# B&R Automation Studio project DuctLines (part 12)

#### Cyclic.ld
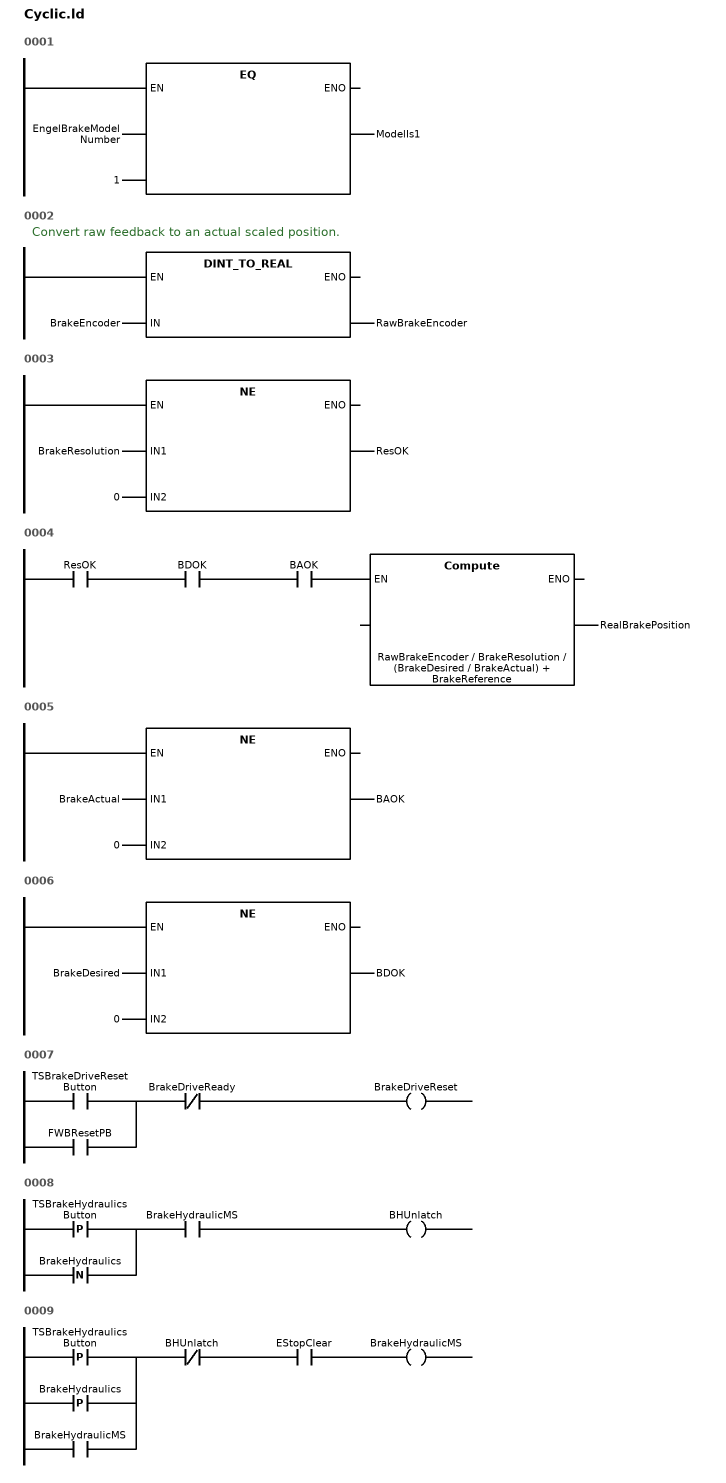
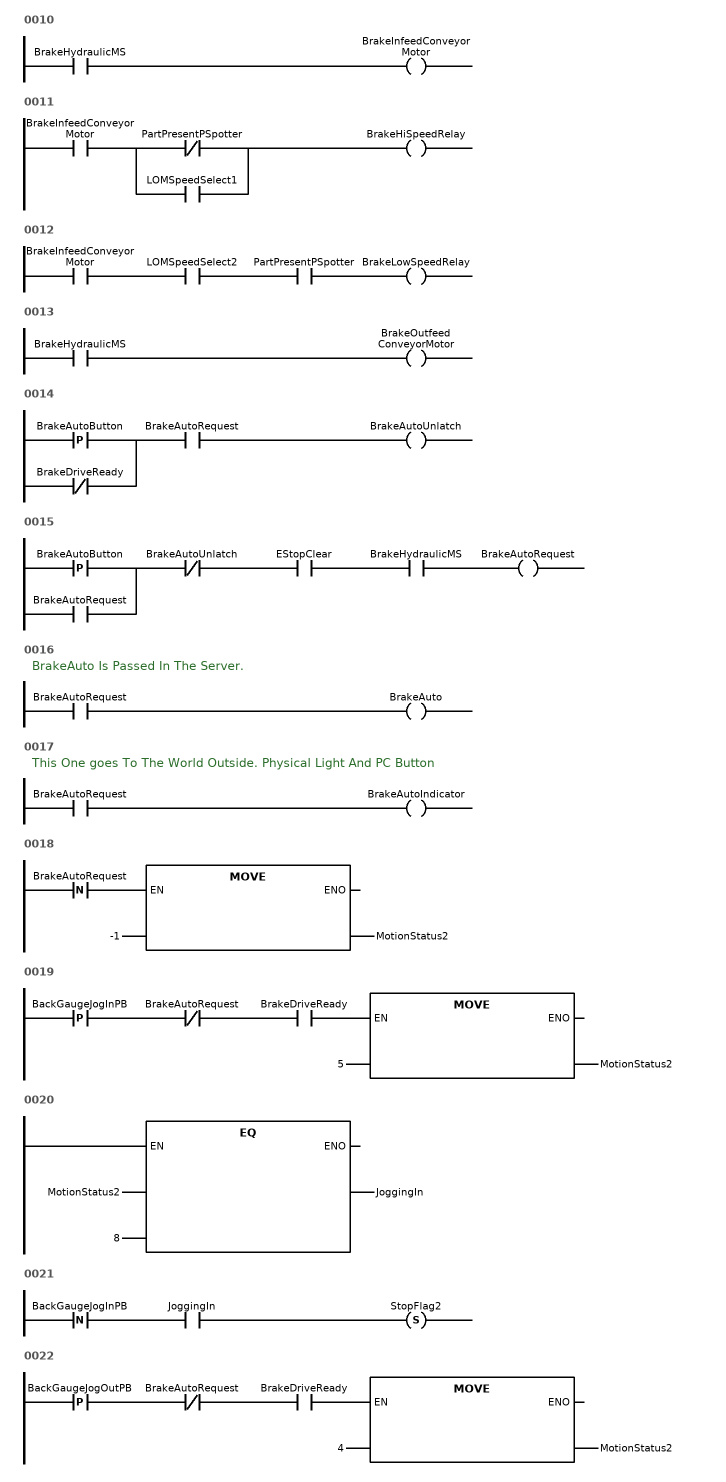
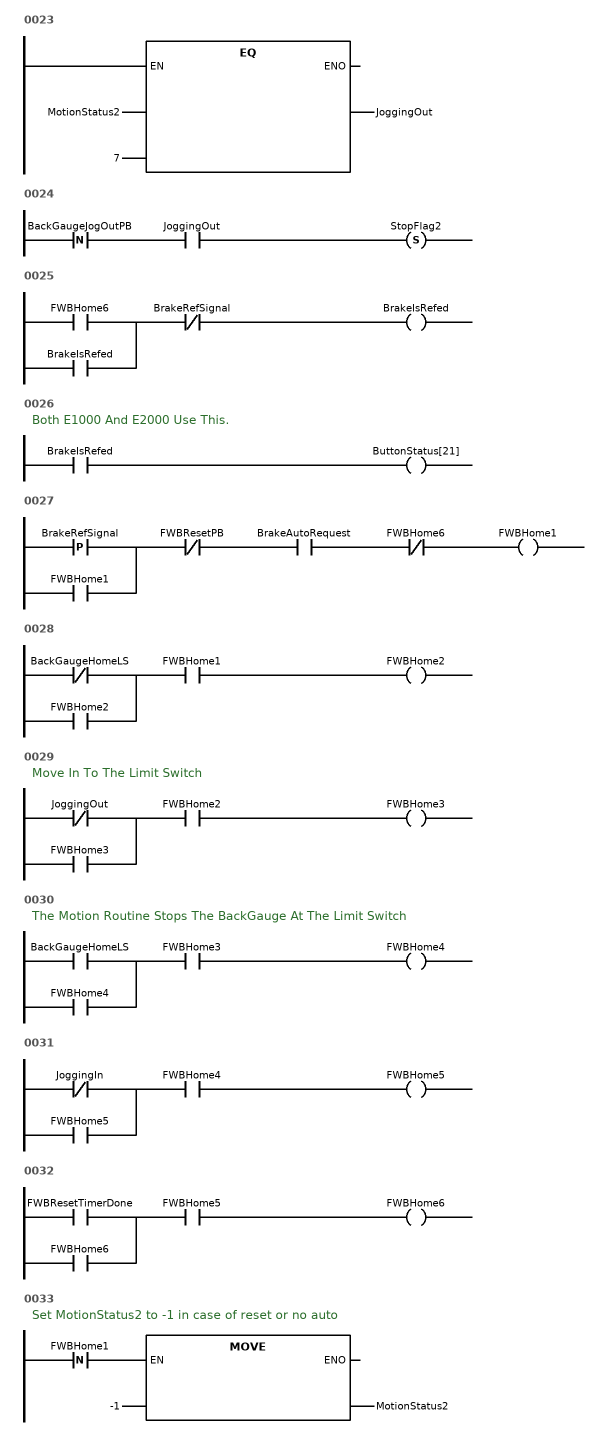
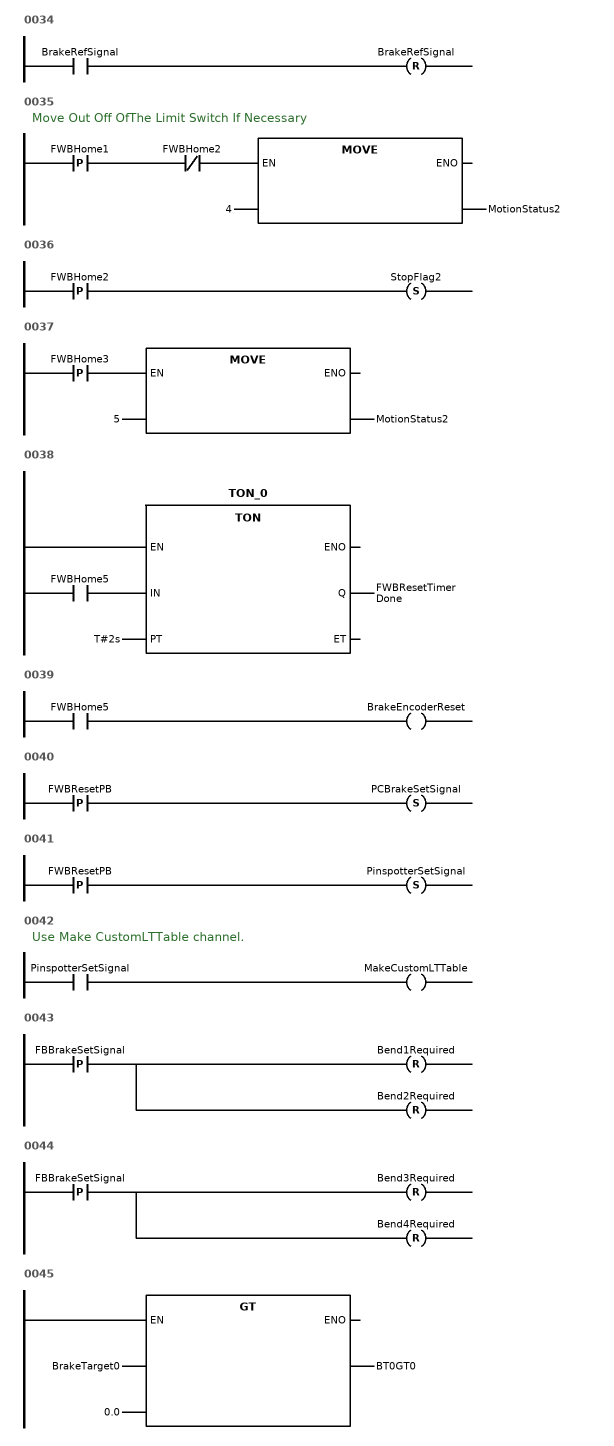
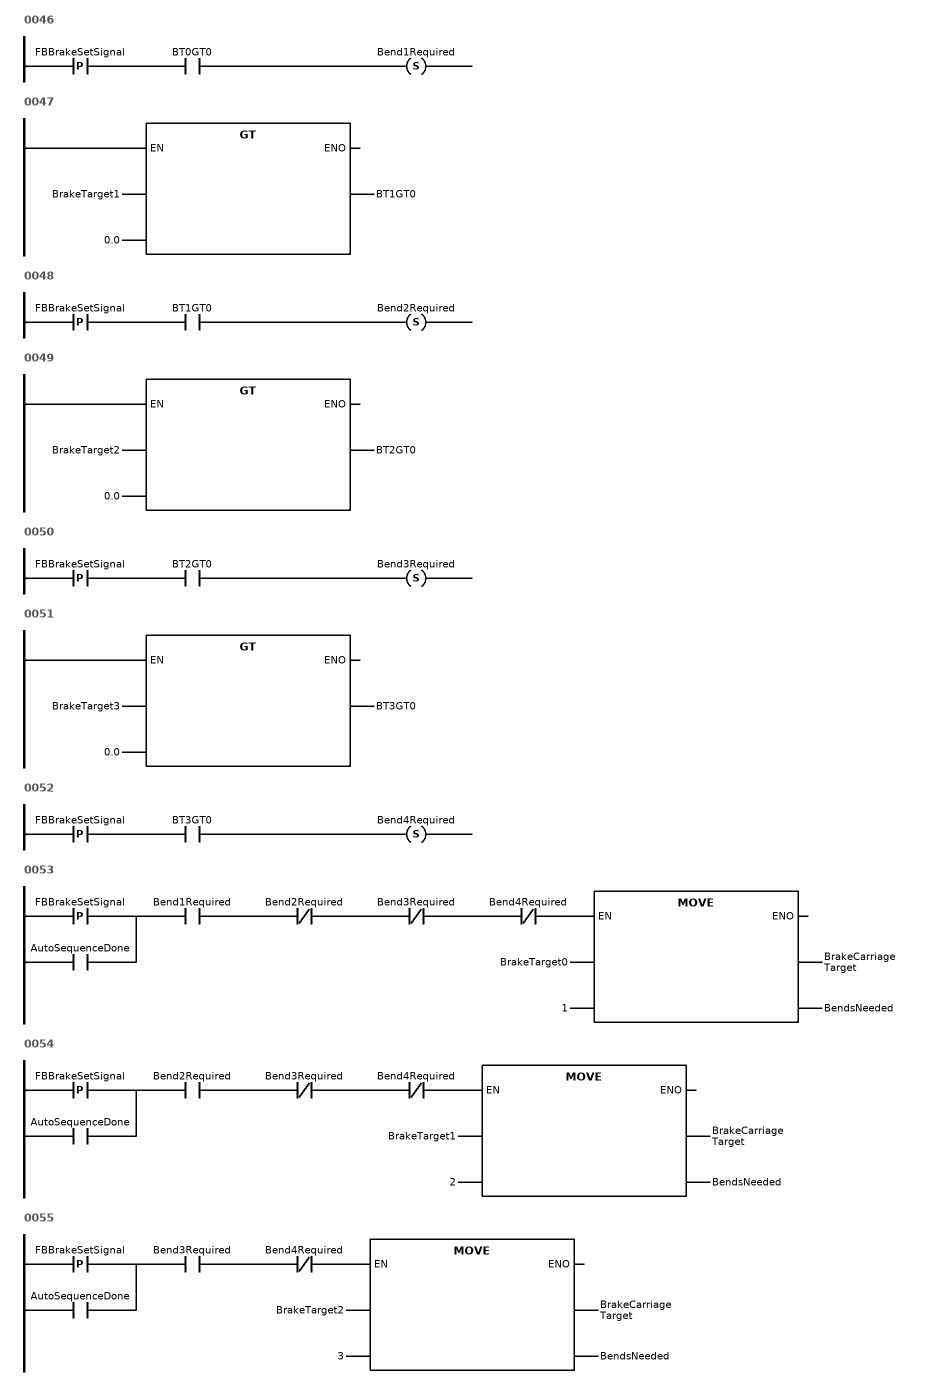
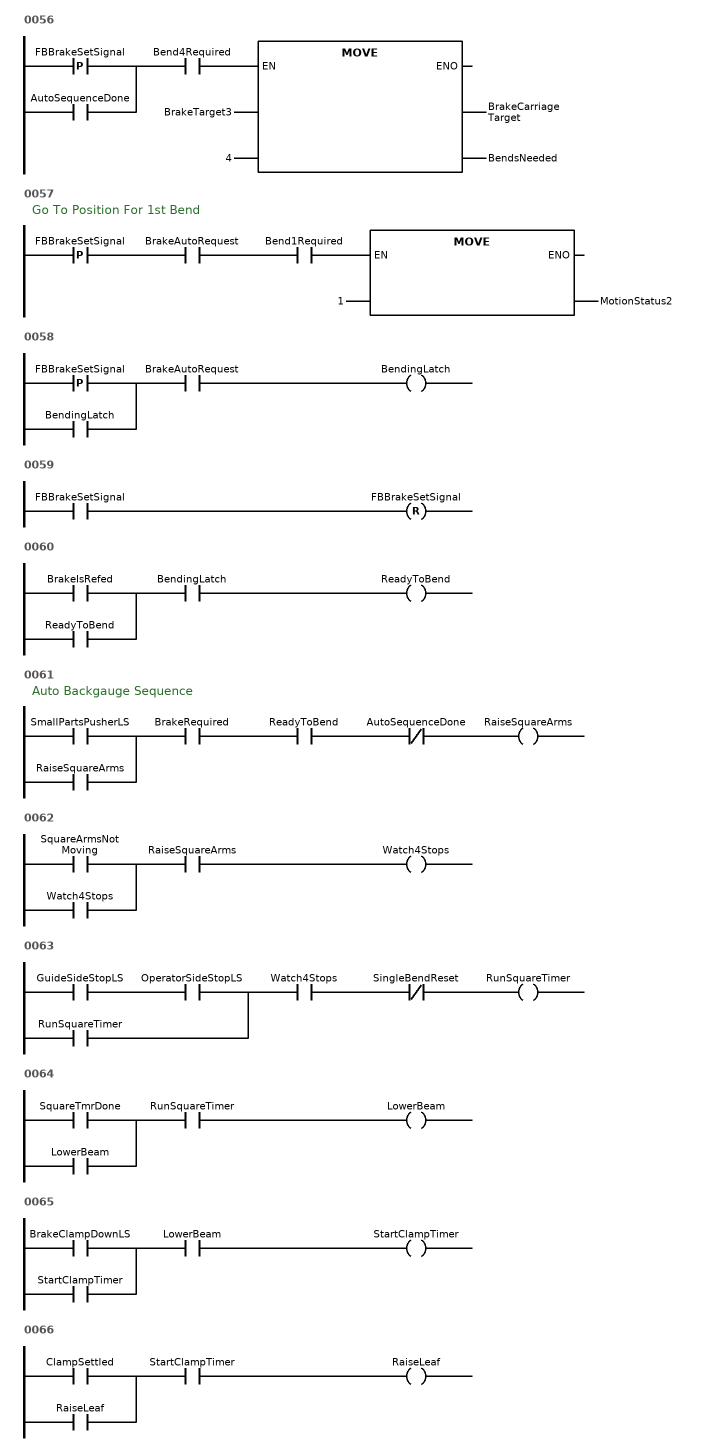
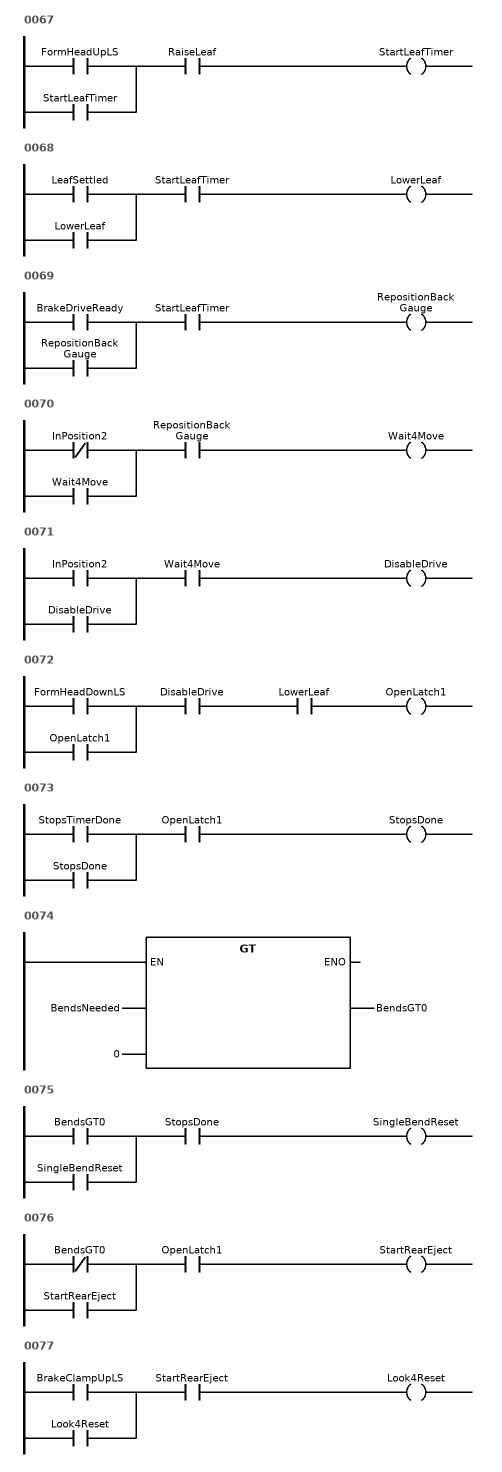
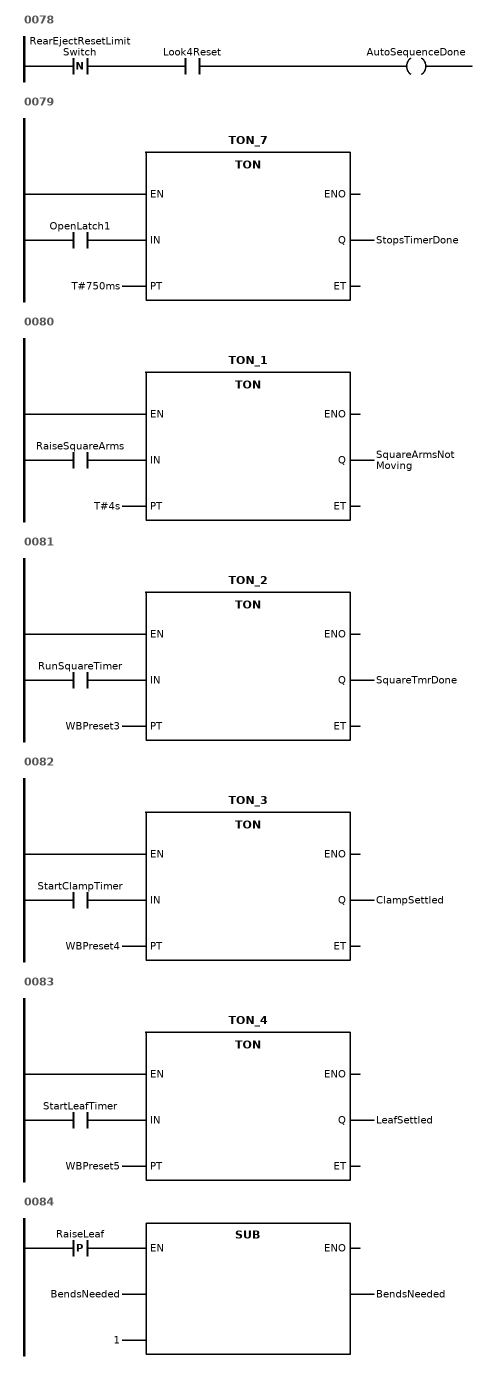
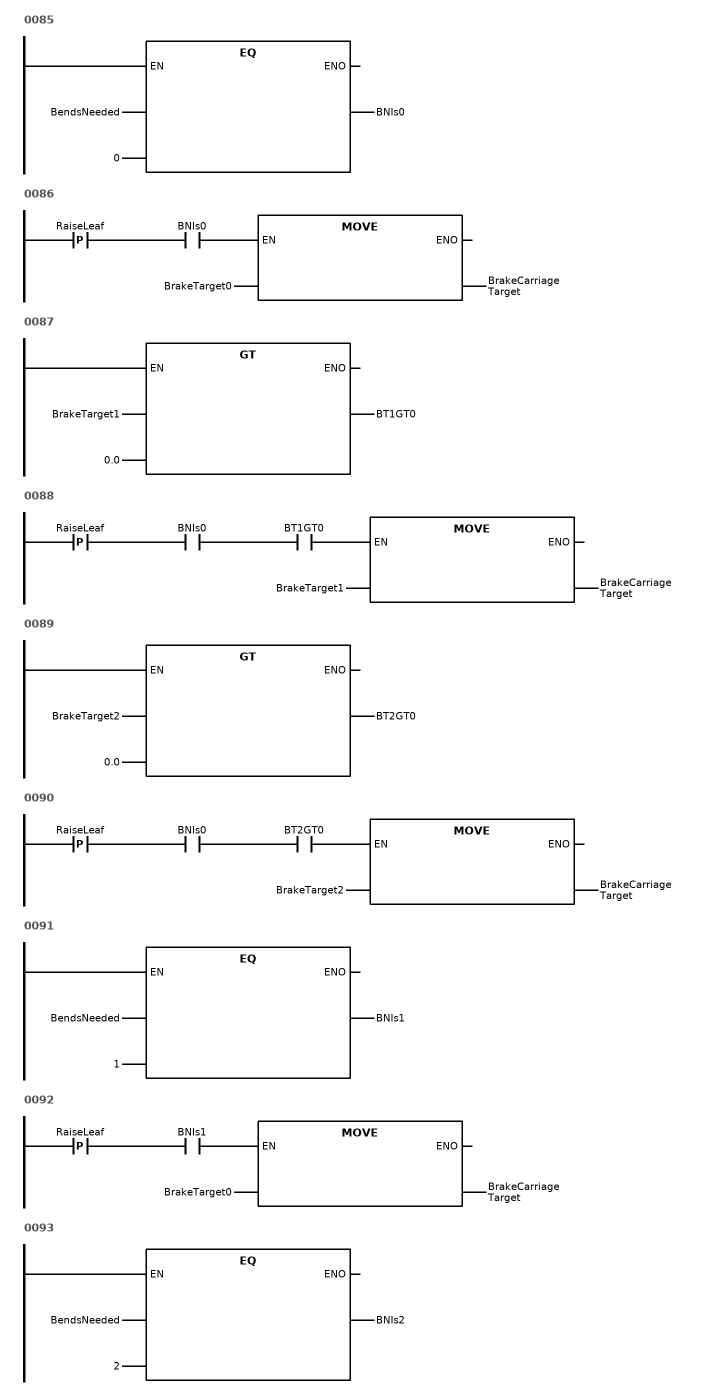
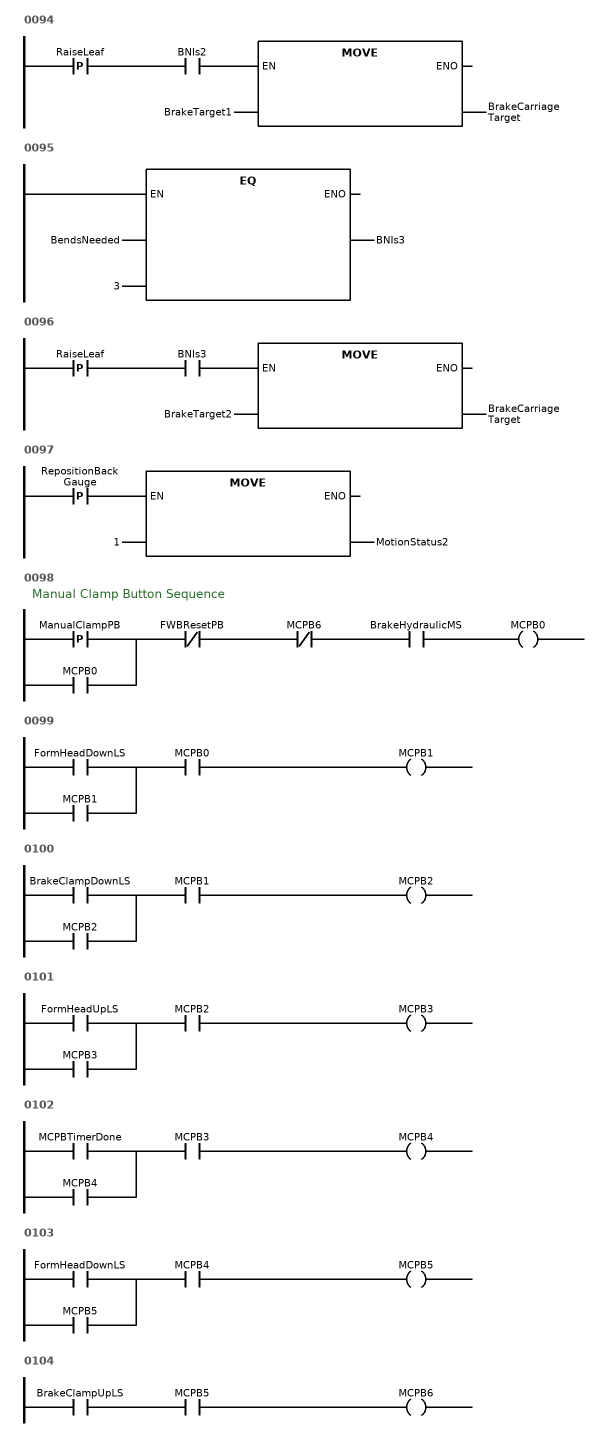
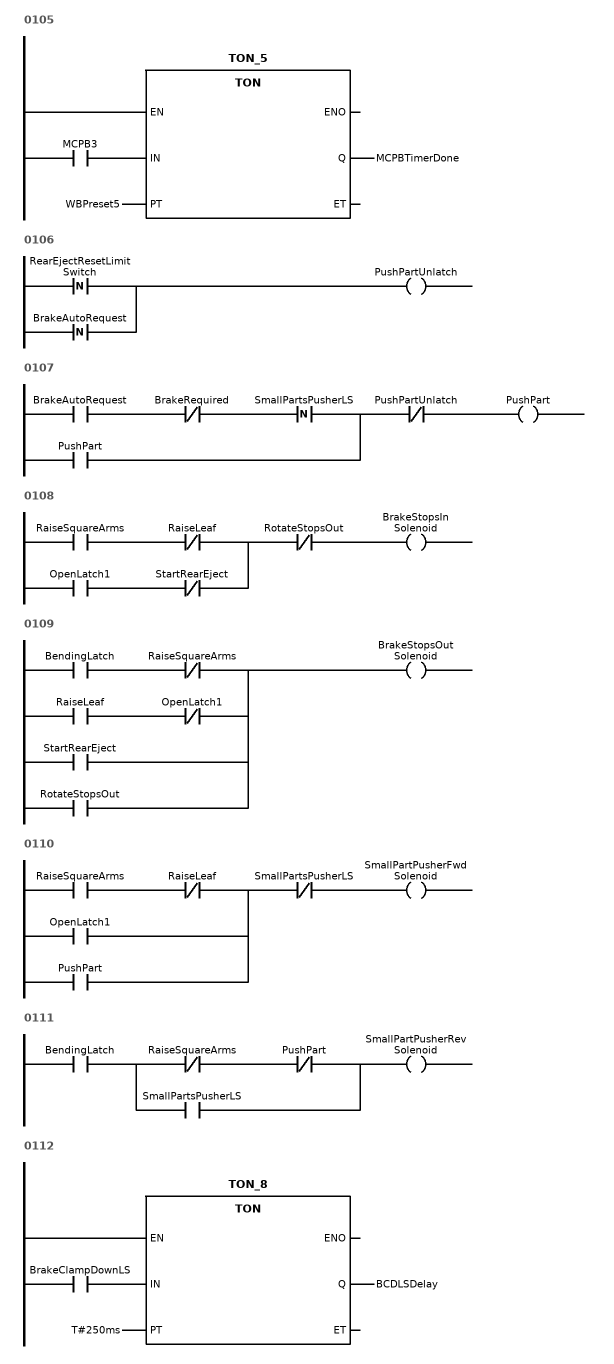
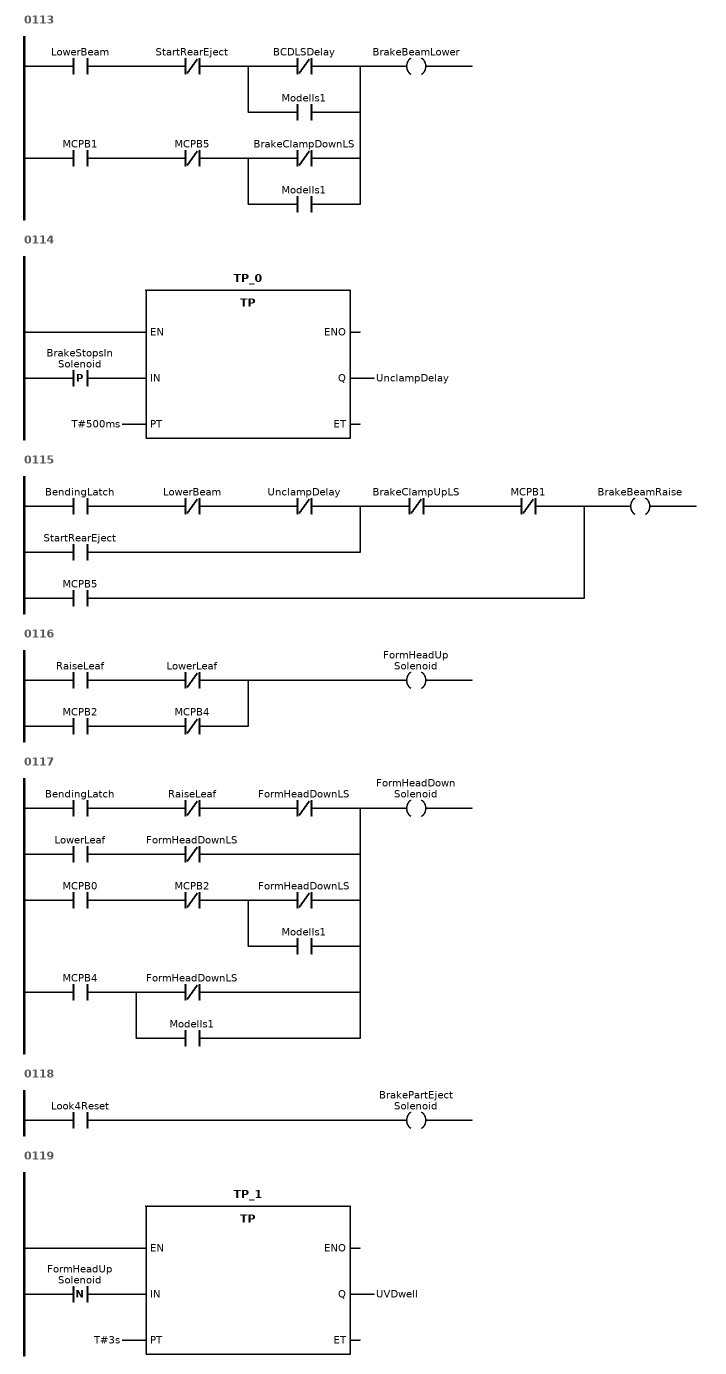
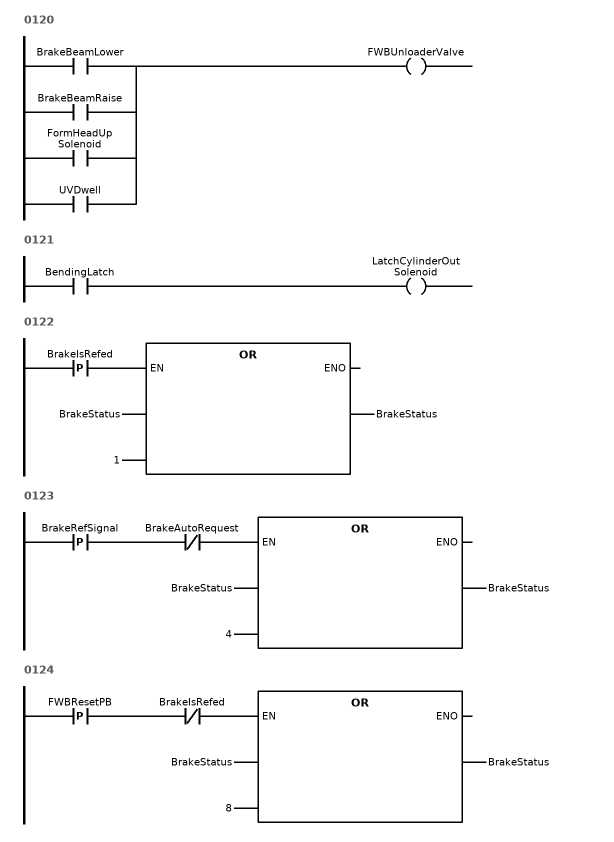
Ladder, written as Structured Text:
```iecst
PROGRAM _CYCLIC
VAR
    _e1 : R_TRIG;
    _e2 : F_TRIG;
    _e3 : R_TRIG;
    _e4 : R_TRIG;
    _e5 : R_TRIG;
    _e6 : R_TRIG;
    _e7 : F_TRIG;
    _e8 : R_TRIG;
    _e9 : F_TRIG;
    _e10 : R_TRIG;
    _e11 : F_TRIG;
    _e12 : R_TRIG;
    _e13 : F_TRIG;
    _e14 : R_TRIG;
    _e15 : R_TRIG;
    _e16 : R_TRIG;
    _e17 : R_TRIG;
    _e18 : R_TRIG;
    _e19 : R_TRIG;
    _e20 : R_TRIG;
    _e21 : R_TRIG;
    _e22 : R_TRIG;
    _e23 : R_TRIG;
    _e24 : R_TRIG;
    _e25 : R_TRIG;
    _p26 : BOOL;
    _e27 : R_TRIG;
    _p28 : BOOL;
    _e29 : R_TRIG;
    _p30 : BOOL;
    _e31 : R_TRIG;
    _e32 : R_TRIG;
    _e33 : R_TRIG;
    _e34 : F_TRIG;
    _e35 : R_TRIG;
    _e36 : R_TRIG;
    _e37 : R_TRIG;
    _e38 : R_TRIG;
    _e39 : R_TRIG;
    _e40 : R_TRIG;
    _e41 : R_TRIG;
    _e42 : R_TRIG;
    _e43 : R_TRIG;
    _e44 : F_TRIG;
    _e45 : F_TRIG;
    _e46 : F_TRIG;
    _e47 : R_TRIG;
    _e48 : F_TRIG;
    _e49 : R_TRIG;
    _e50 : R_TRIG;
    _e51 : R_TRIG;
END_VAR
(* Network 1 *)
ModelIs1 := EngelBrakeModelNumber = 1;

(* Network 2: Convert raw feedback to an actual scaled position. *)
RawBrakeEncoder := DINT_TO_REAL(BrakeEncoder);

(* Network 3 *)
ResOK := BrakeResolution <> 0;

(* Network 4 *)
IF ResOK AND BDOK AND BAOK THEN
    RealBrakePosition := RawBrakeEncoder / BrakeResolution / (BrakeDesired / BrakeActual) + BrakeReference;
END_IF;

(* Network 5 *)
BAOK := BrakeActual <> 0;

(* Network 6 *)
BDOK := BrakeDesired <> 0;

(* Network 7 *)
BrakeDriveReset := (TSBrakeDriveResetButton OR FWBResetPB) AND NOT BrakeDriveReady;

(* Network 8 *)
_e1(CLK := TSBrakeHydraulicsButton);
_e2(CLK := BrakeHydraulics);
BHUnlatch := (_e1.Q OR _e2.Q) AND BrakeHydraulicMS;

(* Network 9 *)
_e3(CLK := TSBrakeHydraulicsButton);
_e4(CLK := BrakeHydraulics);
BrakeHydraulicMS := (_e3.Q OR _e4.Q OR BrakeHydraulicMS) AND NOT BHUnlatch AND EStopClear;

(* Network 10 *)
BrakeInfeedConveyorMotor := BrakeHydraulicMS;

(* Network 11 *)
BrakeHiSpeedRelay := BrakeInfeedConveyorMotor AND (NOT PartPresentPSpotter OR LOMSpeedSelect1);

(* Network 12 *)
BrakeLowSpeedRelay := BrakeInfeedConveyorMotor AND LOMSpeedSelect2 AND PartPresentPSpotter;

(* Network 13 *)
BrakeOutfeedConveyorMotor := BrakeHydraulicMS;

(* Network 14 *)
_e5(CLK := BrakeAutoButton);
BrakeAutoUnlatch := (_e5.Q OR NOT BrakeDriveReady) AND BrakeAutoRequest;

(* Network 15 *)
_e6(CLK := BrakeAutoButton);
BrakeAutoRequest := (_e6.Q OR BrakeAutoRequest) AND NOT BrakeAutoUnlatch AND EStopClear AND BrakeHydraulicMS;

(* Network 16: BrakeAuto Is Passed In The Server. *)
BrakeAuto := BrakeAutoRequest;

(* Network 17: This One goes To The World Outside. Physical Light And PC Button *)
BrakeAutoIndicator := BrakeAutoRequest;

(* Network 18 *)
_e7(CLK := BrakeAutoRequest);
IF _e7.Q THEN MotionStatus2 := -1; END_IF;

(* Network 19 *)
_e8(CLK := BackGaugeJogInPB);
IF _e8.Q AND NOT BrakeAutoRequest AND BrakeDriveReady THEN MotionStatus2 := 5; END_IF;

(* Network 20 *)
JoggingIn := MotionStatus2 = 8;

(* Network 21 *)
_e9(CLK := BackGaugeJogInPB);
IF _e9.Q AND JoggingIn THEN StopFlag2 := TRUE; END_IF;

(* Network 22 *)
_e10(CLK := BackGaugeJogOutPB);
IF _e10.Q AND NOT BrakeAutoRequest AND BrakeDriveReady THEN MotionStatus2 := 4; END_IF;

(* Network 23 *)
JoggingOut := MotionStatus2 = 7;

(* Network 24 *)
_e11(CLK := BackGaugeJogOutPB);
IF _e11.Q AND JoggingOut THEN StopFlag2 := TRUE; END_IF;

(* Network 25 *)
BrakeIsRefed := (FWBHome6 OR BrakeIsRefed) AND NOT BrakeRefSignal;

(* Network 26: Both E1000 And E2000 Use This. *)
ButtonStatus[21] := BrakeIsRefed;

(* Network 27 *)
_e12(CLK := BrakeRefSignal);
FWBHome1 := (_e12.Q OR FWBHome1) AND NOT FWBResetPB AND BrakeAutoRequest AND NOT FWBHome6;

(* Network 28 *)
FWBHome2 := (NOT BackGaugeHomeLS OR FWBHome2) AND FWBHome1;

(* Network 29: Move In To The Limit Switch *)
FWBHome3 := (NOT JoggingOut OR FWBHome3) AND FWBHome2;

(* Network 30: The Motion Routine Stops The BackGauge At The Limit Switch *)
FWBHome4 := (BackGaugeHomeLS OR FWBHome4) AND FWBHome3;

(* Network 31 *)
FWBHome5 := (NOT JoggingIn OR FWBHome5) AND FWBHome4;

(* Network 32 *)
FWBHome6 := (FWBResetTimerDone OR FWBHome6) AND FWBHome5;

(* Network 33: Set MotionStatus2 to -1 in case of reset or no auto *)
_e13(CLK := FWBHome1);
IF _e13.Q THEN MotionStatus2 := -1; END_IF;

(* Network 34 *)
IF BrakeRefSignal THEN BrakeRefSignal := FALSE; END_IF;

(* Network 35: Move Out Off OfThe Limit Switch If Necessary *)
_e14(CLK := FWBHome1);
IF _e14.Q AND NOT FWBHome2 THEN MotionStatus2 := 4; END_IF;

(* Network 36 *)
_e15(CLK := FWBHome2);
IF _e15.Q THEN StopFlag2 := TRUE; END_IF;

(* Network 37 *)
_e16(CLK := FWBHome3);
IF _e16.Q THEN MotionStatus2 := 5; END_IF;

(* Network 38 *)
TON_0(IN := FWBHome5, PT := T#2s);
FWBResetTimerDone := TON_0.Q;

(* Network 39 *)
BrakeEncoderReset := FWBHome5;

(* Network 40 *)
_e17(CLK := FWBResetPB);
IF _e17.Q THEN PCBrakeSetSignal := TRUE; END_IF;

(* Network 41 *)
_e18(CLK := FWBResetPB);
IF _e18.Q THEN PinspotterSetSignal := TRUE; END_IF;

(* Network 42: Use Make CustomLTTable channel. *)
MakeCustomLTTable := PinspotterSetSignal;

(* Network 43 *)
_e19(CLK := FBBrakeSetSignal);
IF _e19.Q THEN
    Bend1Required := FALSE;
    Bend2Required := FALSE;
END_IF;

(* Network 44 *)
_e20(CLK := FBBrakeSetSignal);
IF _e20.Q THEN
    Bend3Required := FALSE;
    Bend4Required := FALSE;
END_IF;

(* Network 45 *)
BT0GT0 := BrakeTarget0 > 0.0;

(* Network 46 *)
_e21(CLK := FBBrakeSetSignal);
IF _e21.Q AND BT0GT0 THEN Bend1Required := TRUE; END_IF;

(* Network 47 *)
BT1GT0 := BrakeTarget1 > 0.0;

(* Network 48 *)
_e22(CLK := FBBrakeSetSignal);
IF _e22.Q AND BT1GT0 THEN Bend2Required := TRUE; END_IF;

(* Network 49 *)
BT2GT0 := BrakeTarget2 > 0.0;

(* Network 50 *)
_e23(CLK := FBBrakeSetSignal);
IF _e23.Q AND BT2GT0 THEN Bend3Required := TRUE; END_IF;

(* Network 51 *)
BT3GT0 := BrakeTarget3 > 0.0;

(* Network 52 *)
_e24(CLK := FBBrakeSetSignal);
IF _e24.Q AND BT3GT0 THEN Bend4Required := TRUE; END_IF;

(* Network 53 *)
_e25(CLK := FBBrakeSetSignal);
_p26 := (_e25.Q OR AutoSequenceDone) AND Bend1Required AND NOT Bend2Required AND NOT Bend3Required AND NOT Bend4Required;
IF _p26 THEN
    BrakeCarriageTarget := BrakeTarget0;
    BendsNeeded := 1;
END_IF;

(* Network 54 *)
_e27(CLK := FBBrakeSetSignal);
_p28 := (_e27.Q OR AutoSequenceDone) AND Bend2Required AND NOT Bend3Required AND NOT Bend4Required;
IF _p28 THEN
    BrakeCarriageTarget := BrakeTarget1;
    BendsNeeded := 2;
END_IF;

(* Network 55 *)
_e29(CLK := FBBrakeSetSignal);
_p30 := (_e29.Q OR AutoSequenceDone) AND Bend3Required AND NOT Bend4Required;
IF _p30 THEN
    BrakeCarriageTarget := BrakeTarget2;
    BendsNeeded := 3;
END_IF;

(* Network 56 *)
_e31(CLK := FBBrakeSetSignal);
IF (_e31.Q OR AutoSequenceDone) AND Bend4Required THEN
    BrakeCarriageTarget := BrakeTarget3;
    BendsNeeded := 4;
END_IF;

(* Network 57: Go To Position For 1st Bend *)
_e32(CLK := FBBrakeSetSignal);
IF _e32.Q AND BrakeAutoRequest AND Bend1Required THEN MotionStatus2 := 1; END_IF;

(* Network 58 *)
_e33(CLK := FBBrakeSetSignal);
BendingLatch := (_e33.Q OR BendingLatch) AND BrakeAutoRequest;

(* Network 59 *)
IF FBBrakeSetSignal THEN FBBrakeSetSignal := FALSE; END_IF;

(* Network 60 *)
ReadyToBend := (BrakeIsRefed OR ReadyToBend) AND BendingLatch;

(* Network 61: Auto Backgauge Sequence *)
RaiseSquareArms := (SmallPartsPusherLS OR RaiseSquareArms) AND BrakeRequired AND ReadyToBend AND NOT AutoSequenceDone;

(* Network 62 *)
Watch4Stops := (SquareArmsNotMoving OR Watch4Stops) AND RaiseSquareArms;

(* Network 63 *)
RunSquareTimer := ((GuideSideStopLS AND OperatorSideStopLS) OR RunSquareTimer) AND Watch4Stops AND NOT SingleBendReset;

(* Network 64 *)
LowerBeam := (SquareTmrDone OR LowerBeam) AND RunSquareTimer;

(* Network 65 *)
StartClampTimer := (BrakeClampDownLS OR StartClampTimer) AND LowerBeam;

(* Network 66 *)
RaiseLeaf := (ClampSettled OR RaiseLeaf) AND StartClampTimer;

(* Network 67 *)
StartLeafTimer := (FormHeadUpLS OR StartLeafTimer) AND RaiseLeaf;

(* Network 68 *)
LowerLeaf := (LeafSettled OR LowerLeaf) AND StartLeafTimer;

(* Network 69 *)
RepositionBackGauge := (BrakeDriveReady OR RepositionBackGauge) AND StartLeafTimer;

(* Network 70 *)
Wait4Move := (NOT InPosition2 OR Wait4Move) AND RepositionBackGauge;

(* Network 71 *)
DisableDrive := (InPosition2 OR DisableDrive) AND Wait4Move;

(* Network 72 *)
OpenLatch1 := (FormHeadDownLS OR OpenLatch1) AND DisableDrive AND LowerLeaf;

(* Network 73 *)
StopsDone := (StopsTimerDone OR StopsDone) AND OpenLatch1;

(* Network 74 *)
BendsGT0 := BendsNeeded > 0;

(* Network 75 *)
SingleBendReset := (BendsGT0 OR SingleBendReset) AND StopsDone;

(* Network 76 *)
StartRearEject := (NOT BendsGT0 OR StartRearEject) AND OpenLatch1;

(* Network 77 *)
Look4Reset := (BrakeClampUpLS OR Look4Reset) AND StartRearEject;

(* Network 78 *)
_e34(CLK := RearEjectResetLimitSwitch);
AutoSequenceDone := _e34.Q AND Look4Reset;

(* Network 79 *)
TON_7(IN := OpenLatch1, PT := T#750ms);
StopsTimerDone := TON_7.Q;

(* Network 80 *)
TON_1(IN := RaiseSquareArms, PT := T#4s);
SquareArmsNotMoving := TON_1.Q;

(* Network 81 *)
TON_2(IN := RunSquareTimer, PT := WBPreset3);
SquareTmrDone := TON_2.Q;

(* Network 82 *)
TON_3(IN := StartClampTimer, PT := WBPreset4);
ClampSettled := TON_3.Q;

(* Network 83 *)
TON_4(IN := StartLeafTimer, PT := WBPreset5);
LeafSettled := TON_4.Q;

(* Network 84 *)
_e35(CLK := RaiseLeaf);
IF _e35.Q THEN BendsNeeded := BendsNeeded - 1; END_IF;

(* Network 85 *)
BNIs0 := BendsNeeded = 0;

(* Network 86 *)
_e36(CLK := RaiseLeaf);
IF _e36.Q AND BNIs0 THEN BrakeCarriageTarget := BrakeTarget0; END_IF;

(* Network 87 *)
BT1GT0 := BrakeTarget1 > 0.0;

(* Network 88 *)
_e37(CLK := RaiseLeaf);
IF _e37.Q AND BNIs0 AND BT1GT0 THEN BrakeCarriageTarget := BrakeTarget1; END_IF;

(* Network 89 *)
BT2GT0 := BrakeTarget2 > 0.0;

(* Network 90 *)
_e38(CLK := RaiseLeaf);
IF _e38.Q AND BNIs0 AND BT2GT0 THEN BrakeCarriageTarget := BrakeTarget2; END_IF;

(* Network 91 *)
BNIs1 := BendsNeeded = 1;

(* Network 92 *)
_e39(CLK := RaiseLeaf);
IF _e39.Q AND BNIs1 THEN BrakeCarriageTarget := BrakeTarget0; END_IF;

(* Network 93 *)
BNIs2 := BendsNeeded = 2;

(* Network 94 *)
_e40(CLK := RaiseLeaf);
IF _e40.Q AND BNIs2 THEN BrakeCarriageTarget := BrakeTarget1; END_IF;

(* Network 95 *)
BNIs3 := BendsNeeded = 3;

(* Network 96 *)
_e41(CLK := RaiseLeaf);
IF _e41.Q AND BNIs3 THEN BrakeCarriageTarget := BrakeTarget2; END_IF;

(* Network 97 *)
_e42(CLK := RepositionBackGauge);
IF _e42.Q THEN MotionStatus2 := 1; END_IF;

(* Network 98: Manual Clamp Button Sequence *)
_e43(CLK := ManualClampPB);
MCPB0 := (_e43.Q OR MCPB0) AND NOT FWBResetPB AND NOT MCPB6 AND BrakeHydraulicMS;

(* Network 99 *)
MCPB1 := (FormHeadDownLS OR MCPB1) AND MCPB0;

(* Network 100 *)
MCPB2 := (BrakeClampDownLS OR MCPB2) AND MCPB1;

(* Network 101 *)
MCPB3 := (FormHeadUpLS OR MCPB3) AND MCPB2;

(* Network 102 *)
MCPB4 := (MCPBTimerDone OR MCPB4) AND MCPB3;

(* Network 103 *)
MCPB5 := (FormHeadDownLS OR MCPB5) AND MCPB4;

(* Network 104 *)
MCPB6 := BrakeClampUpLS AND MCPB5;

(* Network 105 *)
TON_5(IN := MCPB3, PT := WBPreset5);
MCPBTimerDone := TON_5.Q;

(* Network 106 *)
_e44(CLK := RearEjectResetLimitSwitch);
_e45(CLK := BrakeAutoRequest);
PushPartUnlatch := _e44.Q OR _e45.Q;

(* Network 107 *)
_e46(CLK := SmallPartsPusherLS);
PushPart := ((BrakeAutoRequest AND NOT BrakeRequired AND _e46.Q) OR PushPart) AND NOT PushPartUnlatch;

(* Network 108 *)
BrakeStopsInSolenoid := ((RaiseSquareArms AND NOT RaiseLeaf) OR (OpenLatch1 AND NOT StartRearEject)) AND NOT RotateStopsOut;

(* Network 109 *)
BrakeStopsOutSolenoid := (BendingLatch AND NOT RaiseSquareArms) OR (RaiseLeaf AND NOT OpenLatch1) OR StartRearEject OR RotateStopsOut;

(* Network 110 *)
SmallPartPusherFwdSolenoid := ((RaiseSquareArms AND NOT RaiseLeaf) OR OpenLatch1 OR PushPart) AND NOT SmallPartsPusherLS;

(* Network 111 *)
SmallPartPusherRevSolenoid := BendingLatch AND ((NOT RaiseSquareArms AND NOT PushPart) OR SmallPartsPusherLS);

(* Network 112 *)
TON_8(IN := BrakeClampDownLS, PT := T#250ms);
BCDLSDelay := TON_8.Q;

(* Network 113 *)
BrakeBeamLower := (LowerBeam AND NOT StartRearEject AND (NOT BCDLSDelay OR ModelIs1)) OR (MCPB1 AND NOT MCPB5 AND (NOT BrakeClampDownLS OR ModelIs1));

(* Network 114 *)
_e47(CLK := BrakeStopsInSolenoid);
TP_0(IN := _e47.Q, PT := T#500ms);
UnclampDelay := TP_0.Q;

(* Network 115 *)
BrakeBeamRaise := (((BendingLatch AND NOT LowerBeam AND NOT UnclampDelay) OR StartRearEject) AND NOT BrakeClampUpLS AND NOT MCPB1) OR MCPB5;

(* Network 116 *)
FormHeadUpSolenoid := (RaiseLeaf AND NOT LowerLeaf) OR (MCPB2 AND NOT MCPB4);

(* Network 117 *)
FormHeadDownSolenoid := (BendingLatch AND NOT RaiseLeaf AND NOT FormHeadDownLS) OR (LowerLeaf AND NOT FormHeadDownLS) OR (MCPB0 AND NOT MCPB2 AND (NOT FormHeadDownLS OR ModelIs1)) OR (MCPB4 AND (NOT FormHeadDownLS OR ModelIs1));

(* Network 118 *)
BrakePartEjectSolenoid := Look4Reset;

(* Network 119 *)
_e48(CLK := FormHeadUpSolenoid);
TP_1(IN := _e48.Q, PT := T#3s);
UVDwell := TP_1.Q;

(* Network 120 *)
FWBUnloaderValve := BrakeBeamLower OR BrakeBeamRaise OR FormHeadUpSolenoid OR UVDwell;

(* Network 121 *)
LatchCylinderOutSolenoid := BendingLatch;

(* Network 122 *)
_e49(CLK := BrakeIsRefed);
IF _e49.Q THEN BrakeStatus := BrakeStatus OR 1; END_IF;

(* Network 123 *)
_e50(CLK := BrakeRefSignal);
IF _e50.Q AND NOT BrakeAutoRequest THEN BrakeStatus := BrakeStatus OR 4; END_IF;

(* Network 124 *)
_e51(CLK := FWBResetPB);
IF _e51.Q AND NOT BrakeIsRefed THEN BrakeStatus := BrakeStatus OR 8; END_IF;
END_PROGRAM
```

#### Init.ld
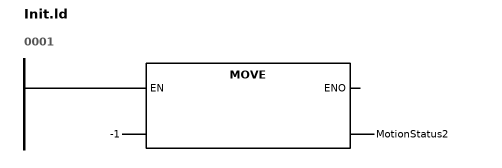
Ladder, written as Structured Text:
```iecst
PROGRAM _INIT
(* Network 1 *)
MotionStatus2 := -1;
END_PROGRAM
```

### Program Logical/PMaster (IEC)

#### Variables.var
```iecst
VAR
	PunchCurrentSelect : DINT;
	OGResult : DINT;
	OGLatch : BOOL;
	FourFootCoil : BOOL;
	FiveFootCoil : BOOL;
	SixFootCoil : BOOL;
	FourResult : DINT;
	FFCLatch : BOOL;
	OneResult : DINT;
	OutsideLatch : BOOL;
	DamperResult : DINT;
	DamperLatch : BOOL;
END_VAR
```

#### Cyclic.ld
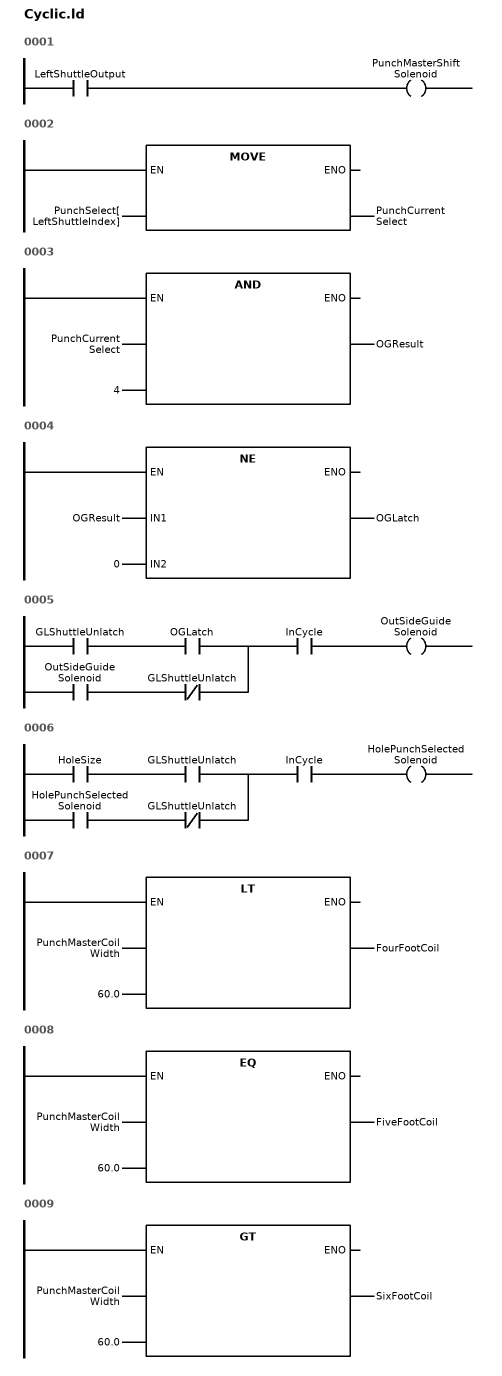
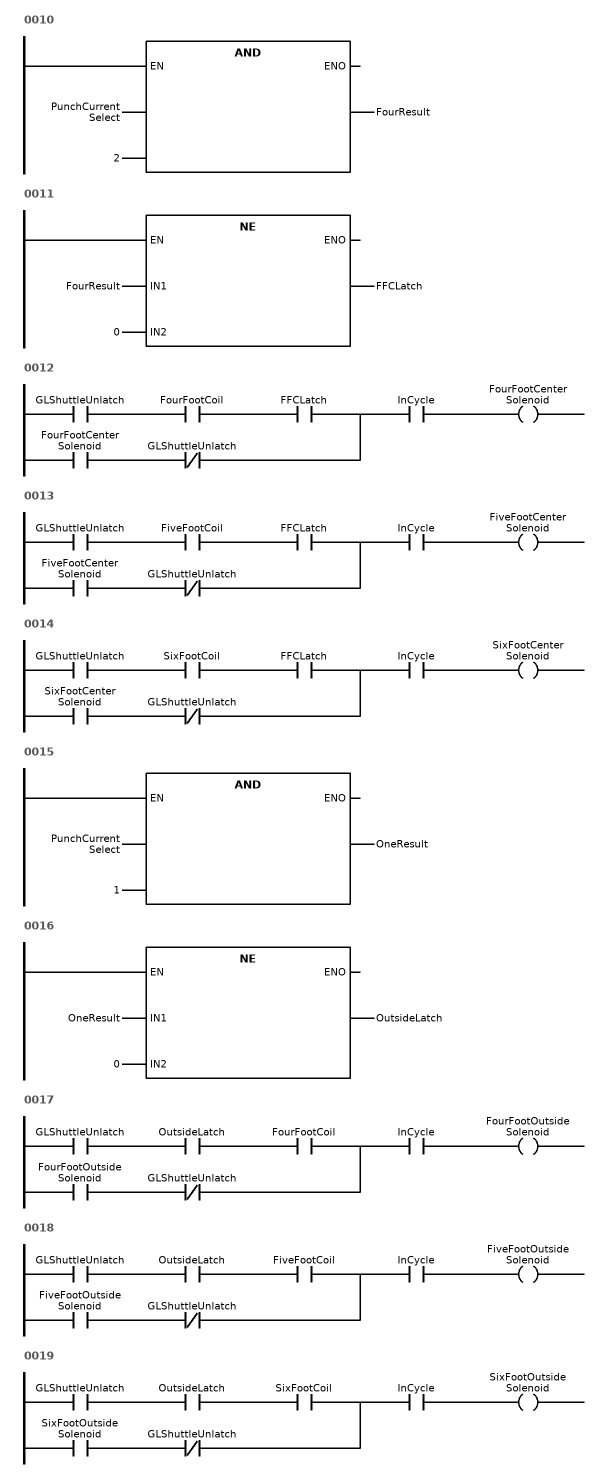
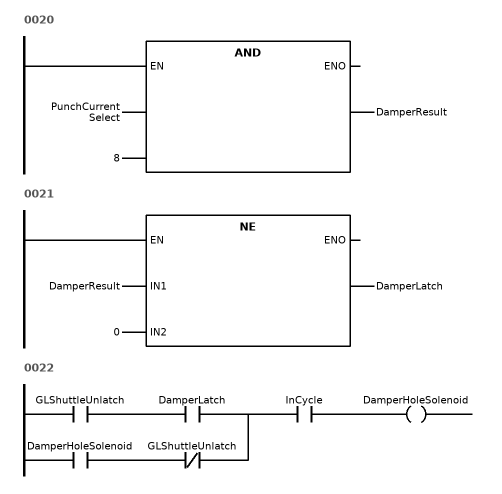
Ladder, written as Structured Text:
```iecst
PROGRAM _CYCLIC
(* Network 1 *)
PunchMasterShiftSolenoid := LeftShuttleOutput;

(* Network 2 *)
PunchCurrentSelect := PunchSelect[LeftShuttleIndex];

(* Network 3 *)
OGResult := PunchCurrentSelect AND 4;

(* Network 4 *)
OGLatch := OGResult <> 0;

(* Network 5 *)
OutSideGuideSolenoid := ((GLShuttleUnlatch AND OGLatch) OR (OutSideGuideSolenoid AND NOT GLShuttleUnlatch)) AND InCycle;

(* Network 6 *)
HolePunchSelectedSolenoid := ((HoleSize AND GLShuttleUnlatch) OR (HolePunchSelectedSolenoid AND NOT GLShuttleUnlatch)) AND InCycle;

(* Network 7 *)
FourFootCoil := PunchMasterCoilWidth < 60.0;

(* Network 8 *)
FiveFootCoil := PunchMasterCoilWidth = 60.0;

(* Network 9 *)
SixFootCoil := PunchMasterCoilWidth > 60.0;

(* Network 10 *)
FourResult := PunchCurrentSelect AND 2;

(* Network 11 *)
FFCLatch := FourResult <> 0;

(* Network 12 *)
FourFootCenterSolenoid := ((GLShuttleUnlatch AND FourFootCoil AND FFCLatch) OR (FourFootCenterSolenoid AND NOT GLShuttleUnlatch)) AND InCycle;

(* Network 13 *)
FiveFootCenterSolenoid := ((GLShuttleUnlatch AND FiveFootCoil AND FFCLatch) OR (FiveFootCenterSolenoid AND NOT GLShuttleUnlatch)) AND InCycle;

(* Network 14 *)
SixFootCenterSolenoid := ((GLShuttleUnlatch AND SixFootCoil AND FFCLatch) OR (SixFootCenterSolenoid AND NOT GLShuttleUnlatch)) AND InCycle;

(* Network 15 *)
OneResult := PunchCurrentSelect AND 1;

(* Network 16 *)
OutsideLatch := OneResult <> 0;

(* Network 17 *)
FourFootOutsideSolenoid := ((GLShuttleUnlatch AND OutsideLatch AND FourFootCoil) OR (FourFootOutsideSolenoid AND NOT GLShuttleUnlatch)) AND InCycle;

(* Network 18 *)
FiveFootOutsideSolenoid := ((GLShuttleUnlatch AND OutsideLatch AND FiveFootCoil) OR (FiveFootOutsideSolenoid AND NOT GLShuttleUnlatch)) AND InCycle;

(* Network 19 *)
SixFootOutsideSolenoid := ((GLShuttleUnlatch AND OutsideLatch AND SixFootCoil) OR (SixFootOutsideSolenoid AND NOT GLShuttleUnlatch)) AND InCycle;

(* Network 20 *)
DamperResult := PunchCurrentSelect AND 8;

(* Network 21 *)
DamperLatch := DamperResult <> 0;

(* Network 22 *)
DamperHoleSolenoid := ((GLShuttleUnlatch AND DamperLatch) OR (DamperHoleSolenoid AND NOT GLShuttleUnlatch)) AND InCycle;
END_PROGRAM
```

### Program Logical/CEF (IEC)

#### Variables.var
```iecst
VAR
	cleat4 : BOOL;
	cleat1 : BOOL;
	cleat2 : BOOL;
	cleat3 : BOOL;
	cleat8 : BOOL;
	cleat5 : BOOL;
	cleat6 : BOOL;
	cleat7 : BOOL;
	TON_0 : TON;
	FirstScan : BOOL;
	TON_10ms_0 : TON_10ms;
	OnTimerDone : BOOL;
	TOF_10ms_0 : TOF_10ms;
	DetectSignal : BOOL;
END_VAR
```

#### Cyclic.ld
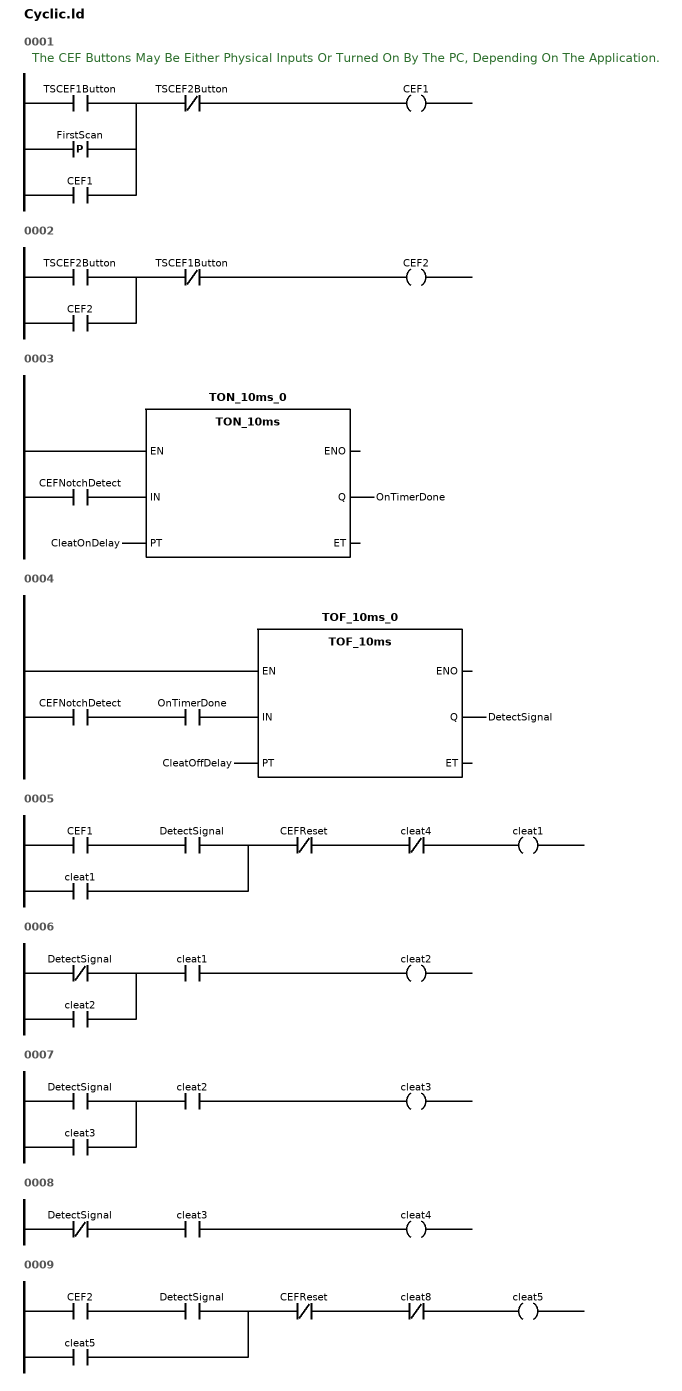
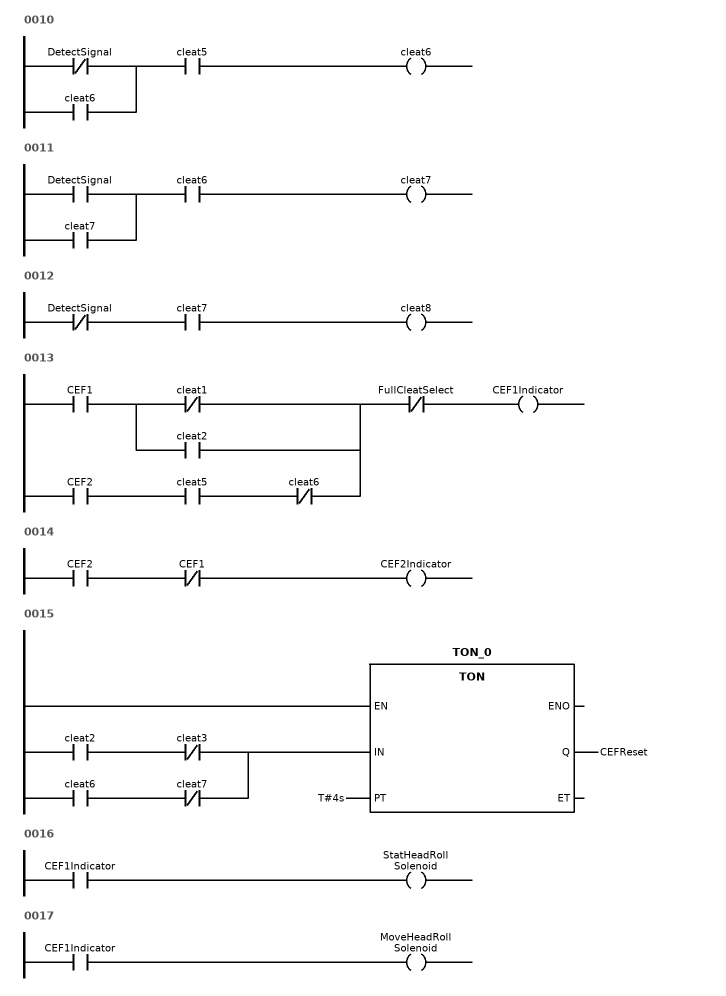
Ladder, written as Structured Text:
```iecst
PROGRAM _CYCLIC
VAR
    _e1 : R_TRIG;
END_VAR
(* Network 1: The CEF Buttons May Be Either Physical Inputs Or Turned On By The PC, Depending On The Application. *)
_e1(CLK := FirstScan);
CEF1 := (TSCEF1Button OR _e1.Q OR CEF1) AND NOT TSCEF2Button;

(* Network 2 *)
CEF2 := (TSCEF2Button OR CEF2) AND NOT TSCEF1Button;

(* Network 3 *)
TON_10ms_0(IN := CEFNotchDetect, PT := CleatOnDelay);
OnTimerDone := TON_10ms_0.Q;

(* Network 4 *)
TOF_10ms_0(IN := CEFNotchDetect AND OnTimerDone, PT := CleatOffDelay);
DetectSignal := TOF_10ms_0.Q;

(* Network 5 *)
cleat1 := ((CEF1 AND DetectSignal) OR cleat1) AND NOT CEFReset AND NOT cleat4;

(* Network 6 *)
cleat2 := (NOT DetectSignal OR cleat2) AND cleat1;

(* Network 7 *)
cleat3 := (DetectSignal OR cleat3) AND cleat2;

(* Network 8 *)
cleat4 := NOT DetectSignal AND cleat3;

(* Network 9 *)
cleat5 := ((CEF2 AND DetectSignal) OR cleat5) AND NOT CEFReset AND NOT cleat8;

(* Network 10 *)
cleat6 := (NOT DetectSignal OR cleat6) AND cleat5;

(* Network 11 *)
cleat7 := (DetectSignal OR cleat7) AND cleat6;

(* Network 12 *)
cleat8 := NOT DetectSignal AND cleat7;

(* Network 13 *)
CEF1Indicator := ((CEF1 AND (NOT cleat1 OR cleat2)) OR (CEF2 AND cleat5 AND NOT cleat6)) AND NOT FullCleatSelect;

(* Network 14 *)
CEF2Indicator := CEF2 AND NOT CEF1;

(* Network 15 *)
TON_0(IN := (cleat2 AND NOT cleat3) OR (cleat6 AND NOT cleat7), PT := T#4s);
CEFReset := TON_0.Q;

(* Network 16 *)
StatHeadRollSolenoid := CEF1Indicator;

(* Network 17 *)
MoveHeadRollSolenoid := CEF1Indicator;
END_PROGRAM
```

#### Init.ld
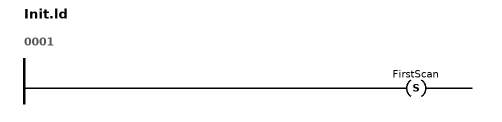
Ladder, written as Structured Text:
```iecst
PROGRAM _INIT
(* Network 1 *)
FirstScan := TRUE;
END_PROGRAM
```

### Program Logical/E2_LOM (IEC)

#### Cyclic.ld
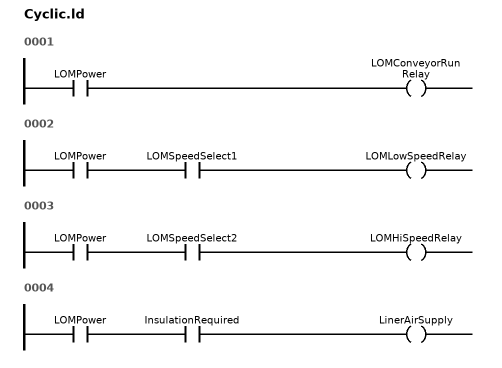
Ladder, written as Structured Text:
```iecst
PROGRAM _CYCLIC
(* Network 1 *)
LOMConveyorRunRelay := LOMPower;

(* Network 2 *)
LOMLowSpeedRelay := LOMPower AND LOMSpeedSelect1;

(* Network 3 *)
LOMHiSpeedRelay := LOMPower AND LOMSpeedSelect2;

(* Network 4 *)
LinerAirSupply := LOMPower AND InsulationRequired;
END_PROGRAM
```

### Program Logical/EFdrHydDrv2 (IEC) - Rungs to control an Engel processor with the original two speed hydraulic solenoids.

#### Variables.var
```iecst
VAR
	difference : DINT;
	AbsoluteDifference : DINT;
	InTargetWindow : BOOL;
	TON_0 : TON;
	MovingToPosition : BOOL;
	MoveInitiated : BOOL;
	PositionLTTarget : BOOL;
	MoveForward : BOOL;
	PositionGTTarget : BOOL;
	MoveReverse : BOOL;
	InSSWindow : BOOL;
	SettleTimerDone : BOOL;
	TP_0 : TP;
	SlowSolenoidDelay : BOOL;
END_VAR
```

#### Cyclic.ld
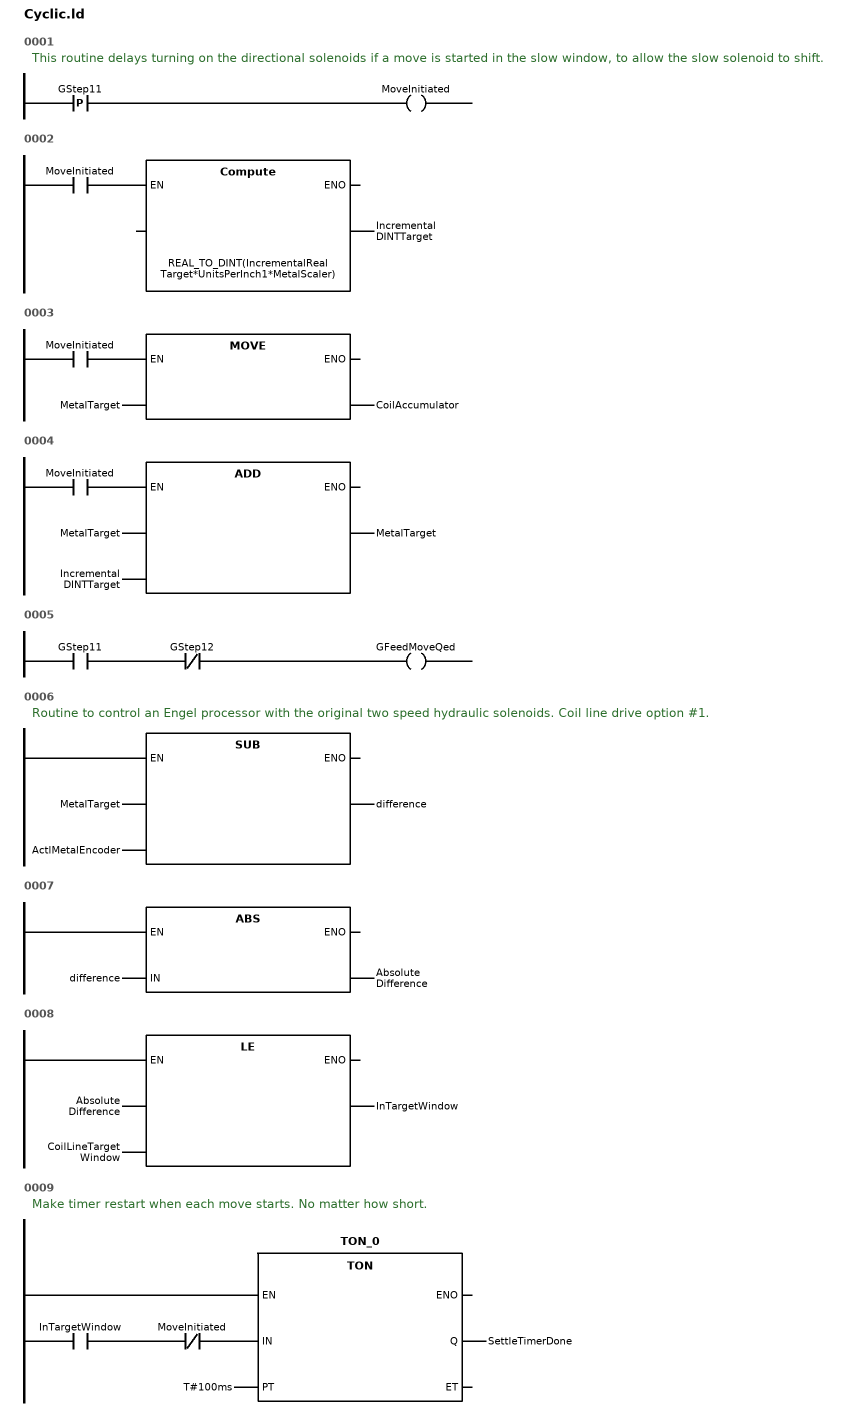
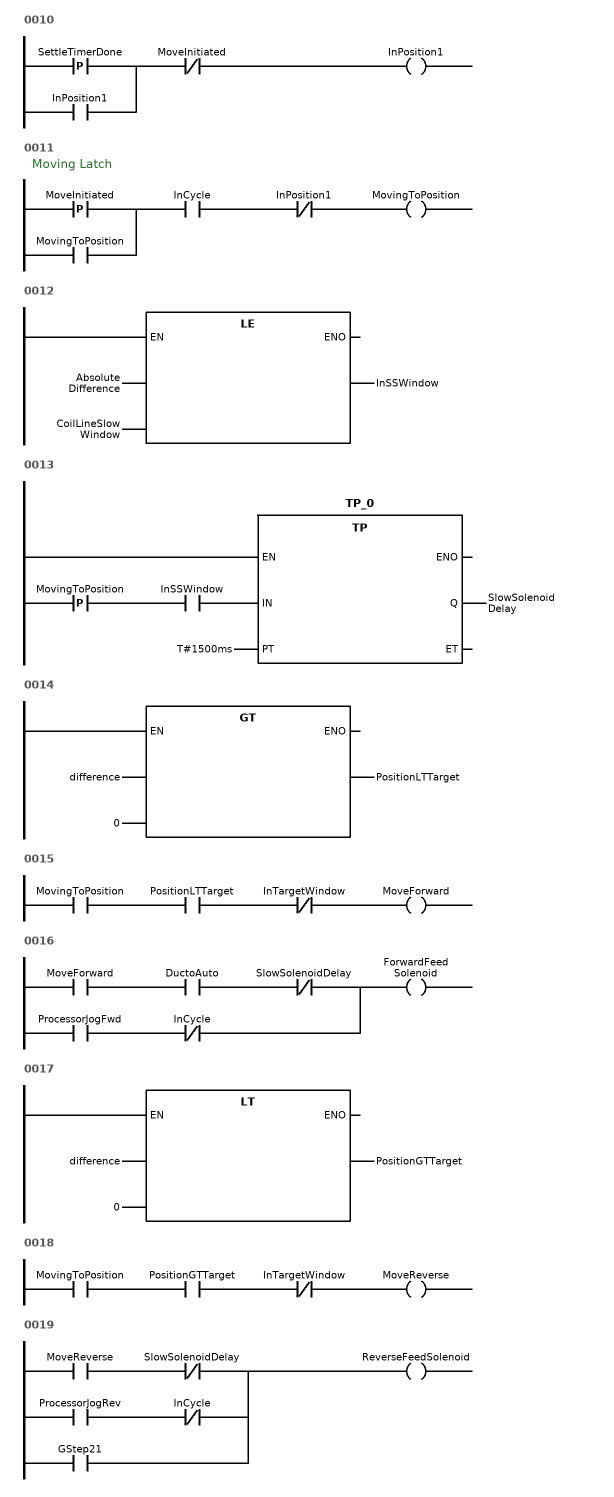
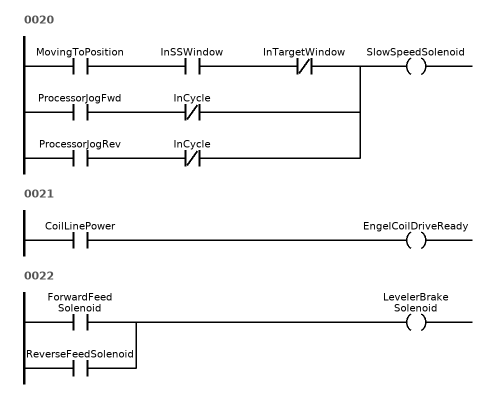
Ladder, written as Structured Text:
```iecst
PROGRAM _CYCLIC
VAR
    _e1 : R_TRIG;
    _e2 : R_TRIG;
    _e3 : R_TRIG;
    _e4 : R_TRIG;
END_VAR
(* Network 1: This routine delays turning on the directional solenoids if a move is started in the slow window, to allow the slow solenoid to shift. *)
_e1(CLK := GStep11);
MoveInitiated := _e1.Q;

(* Network 2 *)
IF MoveInitiated THEN
    IncrementalDINTTarget := REAL_TO_DINT(IncrementalRealTarget*UnitsPerInch1*MetalScaler);
END_IF;

(* Network 3 *)
IF MoveInitiated THEN CoilAccumulator := MetalTarget; END_IF;

(* Network 4 *)
IF MoveInitiated THEN MetalTarget := MetalTarget + IncrementalDINTTarget; END_IF;

(* Network 5 *)
GFeedMoveQed := GStep11 AND NOT GStep12;

(* Network 6: Routine to control an Engel processor with the original two speed hydraulic solenoids. Coil line drive option #1. *)
difference := MetalTarget - ActlMetalEncoder;

(* Network 7 *)
AbsoluteDifference := ABS(difference);

(* Network 8 *)
InTargetWindow := AbsoluteDifference <= CoilLineTargetWindow;

(* Network 9: Make timer restart when each move starts. No matter how short. *)
TON_0(IN := InTargetWindow AND NOT MoveInitiated, PT := T#100ms);
SettleTimerDone := TON_0.Q;

(* Network 10 *)
_e2(CLK := SettleTimerDone);
InPosition1 := (_e2.Q OR InPosition1) AND NOT MoveInitiated;

(* Network 11: Moving Latch *)
_e3(CLK := MoveInitiated);
MovingToPosition := (_e3.Q OR MovingToPosition) AND InCycle AND NOT InPosition1;

(* Network 12 *)
InSSWindow := AbsoluteDifference <= CoilLineSlowWindow;

(* Network 13 *)
_e4(CLK := MovingToPosition);
TP_0(IN := _e4.Q AND InSSWindow, PT := T#1500ms);
SlowSolenoidDelay := TP_0.Q;

(* Network 14 *)
PositionLTTarget := difference > 0;

(* Network 15 *)
MoveForward := MovingToPosition AND PositionLTTarget AND NOT InTargetWindow;

(* Network 16 *)
ForwardFeedSolenoid := (MoveForward AND DuctoAuto AND NOT SlowSolenoidDelay) OR (ProcessorJogFwd AND NOT InCycle);

(* Network 17 *)
PositionGTTarget := difference < 0;

(* Network 18 *)
MoveReverse := MovingToPosition AND PositionGTTarget AND NOT InTargetWindow;

(* Network 19 *)
ReverseFeedSolenoid := (MoveReverse AND NOT SlowSolenoidDelay) OR (ProcessorJogRev AND NOT InCycle) OR GStep21;

(* Network 20 *)
SlowSpeedSolenoid := (MovingToPosition AND InSSWindow AND NOT InTargetWindow) OR (ProcessorJogFwd AND NOT InCycle) OR (ProcessorJogRev AND NOT InCycle);

(* Network 21 *)
EngelCoilDriveReady := CoilLinePower;

(* Network 22 *)
LevelerBrakeSolenoid := ForwardFeedSolenoid OR ReverseFeedSolenoid;
END_PROGRAM
```

### Program Logical/EFeeder (IEC)

#### Variables.var
```iecst
VAR
	AnalogForward : BOOL;
	AnalogReverse : BOOL;
	AutoSignal : BOOL;
	BatchCancelUnlatch : BOOL;
	BeadRollFires : BOOL;
	BeadRollUsedUp : BOOL;
	Block_1 : BOOL;
	BrakeLatch : BOOL;
	ButtonBack7 : BOOL;
	ButtonFires : BOOL;
	ButtonUsedUp : BOOL;
	CenterHoleFires : BOOL;
	CenterHoleTime : TIME;
	CenterHoleUsedUp : BOOL;
	CenterPosA : BOOL;
	CenterShuttleIndex : INT;
	ChangeCShuttle : BOOL;
	ChangeJob1 : BOOL;
	ChangeLShuttle : BOOL;
	ChangeRShuttle : BOOL;
	ClearEncoderSignal : BOOL;
	CleatFires : BOOL;
	CleatUsedUp : BOOL;
	CLPUnlatch : BOOL;
	CShuttleUnlatch : BOOL;
	CustomLTFires : BOOL;
	CustomLTTime : TIME;
	CustomLTUsedUp : BOOL;
	CustomLTValve : BOOL;
	CustomVFires : BOOL;
	CustomVTime : TIME;
	CustomVUsedUp : BOOL;
	DamperLatch : BOOL;
	DamperResult : DINT;
	DataUpdated : BOOL;
	DDDoneTimer : TON;
	DieDelayDone : BOOL;
	DieUpTime : TIME;
	DirectionDelayDone : BOOL;
	DuctoAutoUnlatch : BOOL;
	FeedMoveQed : BOOL;
	FFCLatch : BOOL;
	FiveFootCoil : BOOL;
	FourFootCoil : BOOL;
	FourResult : DINT;
	GapPulse : BOOL;
	GapTP : BOOL;
	GTime : TIME;
	HalfUpdated1 : BOOL;
	HalfUpdated2 : BOOL;
	HolePunchSelecedtSolenoid : BOOL;
	IncPartsMade : BOOL;
	InitMoveSignal : BOOL;
	InPositionBand : REAL := 0.01;
	JobChanging : BOOL;
	LeftHoleFires : BOOL;
	LeftHoleTime : TIME;
	LeftHoleUsedUp : BOOL;
	LeftPosA : BOOL;
	LShuttleUnlatch : BOOL;
	LTFires : BOOL;
	LTTime : TIME;
	LTUsedUp : BOOL;
	ManualSignal : BOOL;
	MarkAccumulator : REAL;
	MetalEncoderLatch : DINT;
	NewRunJobOk : BOOL;
	NextMoveComplete : BOOL;
	NextMoveLookAgain : BOOL;
	NoShearHits : BOOL;
	OGLatch : BOOL;
	OGResult : DINT;
	OneResult : DINT;
	OutsideLatch : BOOL;
	PartCutOff : BOOL;
	PartRefOK : BOOL;
	PunchCurrentSelect : DINT;
	RightHoleFires : BOOL;
	RightHoleTime : TIME;
	RightHoleUsedUp : BOOL;
	RightPosA : BOOL;
	RollEnableUnlatch : BOOL;
	RShuttleUnlatch : BOOL;
	RTotalInches : REAL;
	RunSpeedCalculated : BOOL;
	SetConnectorChange : BOOL;
	ShearBrakeFires : BOOL;
	ShearBrakeUsedUp : BOOL;
	ShearFires : BOOL;
	ShearHitsLTZero : BOOL;
	shearTime : TIME;
	ShearUsedUp : BOOL;
	SixFootCoil : BOOL;
	SmallResult : REAL;
	Step04A : BOOL;
	Step05A : BOOL;
	Step05B : BOOL;
	Step06 : BOOL;
	Step07 : BOOL;
	Step08 : BOOL;
	Step09 : BOOL;
	Step10 : BOOL;
	Step11 : BOOL;
	Step15 : BOOL;
	Step16 : BOOL;
	Step17 : BOOL;
	Step18 : BOOL;
	Step18A : BOOL;
	Step18B : BOOL;
	Step19 : BOOL;
	ThirdOff1 : BOOL;
	ThirdOff2 : BOOL;
	ThirdOff3 : BOOL;
	TON_0 : TON;
	TON_1 : TON;
	TON_10 : TON;
	TON_Warning : TON;
	TP_0 : TP;
	TP_1 : TP;
	TP_2 : TP;
	TP_3 : TP;
	TP_4 : TP;
	TP_5 : TP;
	TP_6 : TP;
	TP_7 : TP;
	TP_8 : TP;
	TP_9 : TP;
	UnlatchBender : BOOL;
	UnlatchButtons : BOOL;
	VFires : BOOL;
	VTime : TIME;
	VUsedUp : BOOL;
	Wait1Ready : BOOL;
	Wait2Ready : BOOL;
	Wait3Ready : BOOL;
	WaitCon1 : BOOL;
	WaitCon2 : BOOL;
	ZCOLT0 : BOOL;
	ZCReverseComplete : BOOL;
	ZCSCTimer : TON;
	ZCSettleComplete : BOOL;
	ZeroCropDifference : DINT;
	ZRCTon : TON;
	FinalScan : BOOL;
	Step12 : BOOL;
	SHLT0 : BOOL;
	Step20 : BOOL;
	ReturnTarget : DINT;
	ReturnComplete : BOOL;
	Step21 : BOOL;
	ReturnCalculated : BOOL;
	Step22 : BOOL;
	JobsDifferent : BOOL;
END_VAR
```
